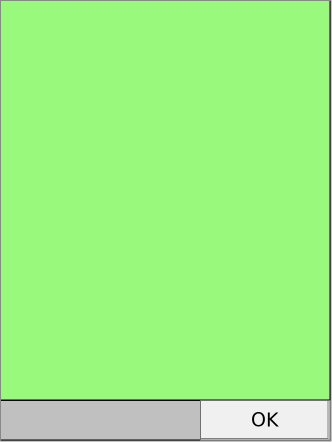
VISUALIZATION V_Dialog_Mob  // 332x442
    Rectangle (0,400 330x40)
    Rectangle (0,0 330x400)
    Button (200,400 130x40), "OK"
        OnMouseUp: change screen: Previous 
END_VISUALIZATION

(* stored: Version 1.1.0.1, ProductVersion 3.1.4018.5
   Visu V_Dialog_Mob: Id {88d8a45c-a534-4a07-aea3-85f4e45470a3} *)
